TYPE machineSettings :
STRUCT
END_STRUCT
END_TYPE

(* stored: Version 1.1.0.1, ProductVersion 3.1.4024.3
   DUT machineSettings: Id {c5788160-e90f-459d-82d6-01fc8aba7eb7} *)
